(* IEC 61131-3 sources: BODAS-HelloWorld/extracted_st/bodas_rc18_12_40/plc_logic/application/02_easyconfig/easyconfig_import/bds_syspb_ec/bds_syspb_ec_gvl, 1 file *)

(* ---- bds_sysPb_ec_gvl.st ---- *)
(* --- Interface --- *)
{attribute 'qualified_only' := ''}
VAR_GLOBAL CONSTANT
    ml290rts_bs_HelloWorld : USINT := bds_sysPb_vrnt_te.bds_sysPb_vrnt01_E;
END_VAR
